{attribute addProperty BoxType "EP3314-0002-0019"}
{attribute addProperty Id "TC_Inputs_ChannelAT %I*ARRAY[0..6] OF TC_Inputs_Channel_F16A160D128160WcStateAT %I*WcState_98A4DF7520.250InfoDataAT %I*InfoData_BC63D37F80100"}
{attribute addProperty CRC "2970462671"}
{attribute addProperty SizeInBites "210"}
{attribute addProperty SizeInBytes "26.25"}
TYPE EP3314_A69716D7 :
STRUCT
	{attribute addProperty Name "TC_Inputs_Channel"}
	TC_Inputs_Channel : ARRAY[0..6] OF TC_Inputs_Channel_F16A160D;
	{attribute addProperty Name "WcState"}
	WcState : WcState_98A4DF75;
	{attribute addProperty Name "InfoData"}
	InfoData : InfoData_BC63D37F;
END_STRUCT
END_TYPE

(* stored: Version 1.2.0.0, ProductVersion 3.1.4024.9
   DUT EP3314_A69716D7: Id {4220fd88-6fe2-4b00-973c-b01f5528fb32} *)
